// TIA Portal project "VFD" (V15)

(* hardware
DEVICE "S7-1200 station_1"  S7-1200 Station
   slot 0: "Rack_0"  S7-1200 Rack  Rack  V1.0
   slot 1: "PLC_1"  CPU 1212C AC/DC/Rly  6ES7 212-1BE40-0XB0  V4.2
*)

// ===== PLC "PLC_1"  CPU 1212C AC/DC/Rly =====

VAR_GLOBAL   // PLC tag table "Default tag table"
   "START" AT %I0.0 : Bool;
   "STOP" AT %I0.1 : Bool;
   "F" AT %Q0.0 : Bool;
   "R" AT %Q0.1 : Bool;
   "15HZ" AT %Q0.2 : Bool;
   "30HZ" AT %Q0.3 : Bool;
   "X" AT %M0.0 : Bool;
   "15HZ F" AT %M0.5 : Bool;
   "30HZ F" AT %M0.3 : Bool;
   "Tag_1" AT %M0.7 : Bool;
   "Tag_2" AT %M7.2 : Bool;
   "3OHZ R" AT %M1.3 : Bool;
   "15HZ R" AT %M1.5 : Bool;
   "Tag_3" AT %M7.4 : Bool;
END_VAR

// folder: System blocks/Program resources

DATA_BLOCK "T1"   // DB1
{ S7_Optimized_Access := 'TRUE' }
AUTHOR : Simatic
FAMILY : IEC
NAME : IEC_TMR
VERSION : 1.0
// stored: InstanceOfName IEC_TIMER
"IEC_TIMER"
BEGIN
END_DATA_BLOCK

DATA_BLOCK "T2"   // DB2
{ S7_Optimized_Access := 'TRUE' }
AUTHOR : Simatic
FAMILY : IEC
NAME : IEC_TMR
VERSION : 1.0
// stored: InstanceOfName IEC_TIMER
"IEC_TIMER"
BEGIN
END_DATA_BLOCK

DATA_BLOCK "T3"   // DB3
{ S7_Optimized_Access := 'TRUE' }
AUTHOR : Simatic
FAMILY : IEC
NAME : IEC_TMR
VERSION : 1.0
// stored: InstanceOfName IEC_TIMER
"IEC_TIMER"
BEGIN
END_DATA_BLOCK

DATA_BLOCK "T4"   // DB4
{ S7_Optimized_Access := 'TRUE' }
AUTHOR : Simatic
FAMILY : IEC
NAME : IEC_TMR
VERSION : 1.0
// stored: InstanceOfName IEC_TIMER
"IEC_TIMER"
BEGIN
END_DATA_BLOCK

DATA_BLOCK "T5"   // DB5
{ S7_Optimized_Access := 'TRUE' }
AUTHOR : Simatic
FAMILY : IEC
NAME : IEC_TMR
VERSION : 1.0
// stored: InstanceOfName IEC_TIMER
"IEC_TIMER"
BEGIN
END_DATA_BLOCK

DATA_BLOCK "T6"   // DB6
{ S7_Optimized_Access := 'TRUE' }
AUTHOR : Simatic
FAMILY : IEC
NAME : IEC_TMR
VERSION : 1.0
// stored: InstanceOfName IEC_TIMER
"IEC_TIMER"
BEGIN
END_DATA_BLOCK

// folder: (top level)

ORGANIZATION_BLOCK "Main"   // OB1, LAD, ProgramCycle
TITLE = "Main Program Sweep (Cycle)"
{ S7_Optimized_Access := 'TRUE' }
VERSION : 0.1
   VAR_INPUT
      Initial_Call : Bool;   // Initial call of this OB
      Remanence : Bool;   // =True, if remanent data are available
   END_VAR
BEGIN

REGION Network 1
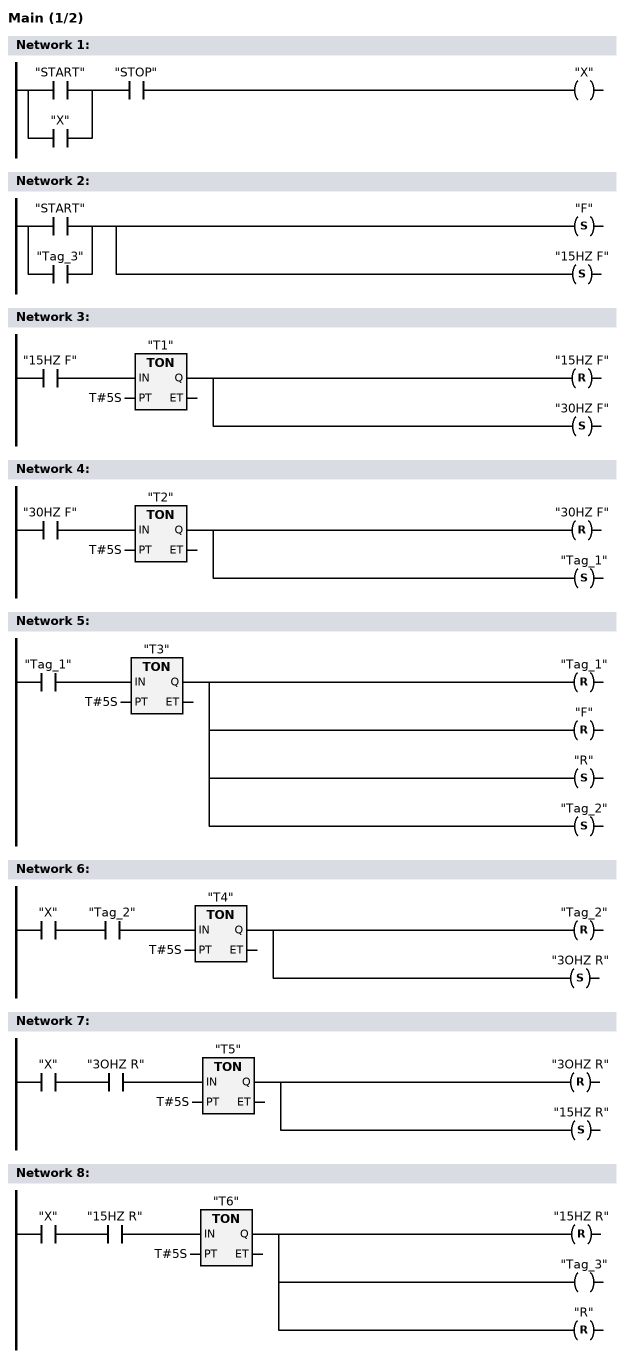
   RUNG wire#powerrail
      Contact( "START" )
      wire#w1
      Contact( "STOP" )
      Coil( "X" )
   END_RUNG
   RUNG wire#powerrail
      Contact( "X" )
   END_RUNG wire#w1
   // the same network as SCL:
   "X" := ("START" OR "X") AND "STOP";
END_REGION

REGION Network 2
   RUNG wire#powerrail
      Contact( "START" )
      wire#w1
      S_Coil( "F" )
   END_RUNG
   RUNG wire#powerrail
      Contact( "Tag_3" )
   END_RUNG wire#w1
   RUNG wire#w1
      S_Coil( "15HZ F" )
   END_RUNG
   // the same network as SCL:
   IF "START" OR "Tag_3" THEN
       "F" := TRUE;
       "15HZ F" := TRUE;
   END_IF;
END_REGION

REGION Network 3
   "T1".TON(IN := "15HZ F", PT := T#5S);
   IF "T1".Q THEN
       "15HZ F" := FALSE;
       "30HZ F" := TRUE;
   END_IF;
END_REGION

REGION Network 4
   "T2".TON(IN := "30HZ F", PT := T#5S);
   IF "T2".Q THEN
       "30HZ F" := FALSE;
       "Tag_1" := TRUE;
   END_IF;
END_REGION

REGION Network 5
   "T3".TON(IN := "Tag_1", PT := T#5S);
   IF "T3".Q THEN
       "Tag_1" := FALSE;
       "F" := FALSE;
       "R" := TRUE;
       "Tag_2" := TRUE;
   END_IF;
END_REGION

REGION Network 6
   "T4".TON(IN := "X" AND "Tag_2", PT := T#5S);
   IF "T4".Q THEN
       "Tag_2" := FALSE;
       "3OHZ R" := TRUE;
   END_IF;
END_REGION

REGION Network 7
   "T5".TON(IN := "X" AND "3OHZ R", PT := T#5S);
   IF "T5".Q THEN
       "3OHZ R" := FALSE;
       "15HZ R" := TRUE;
   END_IF;
END_REGION

REGION Network 8
   "T6".TON(IN := "X" AND "15HZ R", PT := T#5S);
   IF "T6".Q THEN "15HZ R" := FALSE; END_IF;
   "Tag_3" := "T6".Q;
   IF "T6".Q THEN "R" := FALSE; END_IF;
END_REGION

REGION Network 9
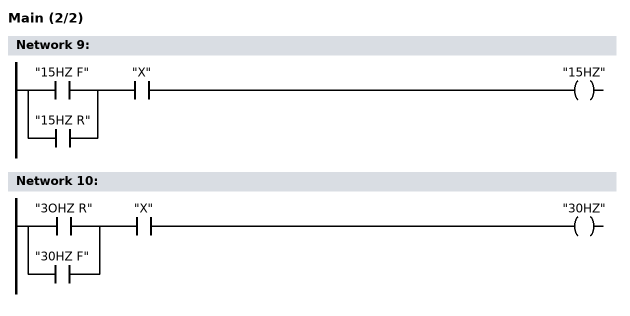
   RUNG wire#powerrail
      Contact( "15HZ F" )
      wire#w1
      Contact( "X" )
      Coil( "15HZ" )
   END_RUNG
   RUNG wire#powerrail
      Contact( "15HZ R" )
   END_RUNG wire#w1
   // the same network as SCL:
   "15HZ" := ("15HZ F" OR "15HZ R") AND "X";
END_REGION

REGION Network 10
   RUNG wire#powerrail
      Contact( "3OHZ R" )
      wire#w1
      Contact( "X" )
      Coil( "30HZ" )
   END_RUNG
   RUNG wire#powerrail
      Contact( "30HZ F" )
   END_RUNG wire#w1
   // the same network as SCL:
   "30HZ" := ("3OHZ R" OR "30HZ F") AND "X";
END_REGION
END_ORGANIZATION_BLOCK